	FUNCTION_BLOCK FB 1042
	TITLE =A_2914_MXZ01MA BELT CONVEYOR 4600 GERM 3
	//COPYRIGHT:     (C) 2009  BUHLER AG, CH-9240 UZWIL, SWITZERLAND
	//
	//PRODUCT:       WinCoS_BIW01_09
	//
	//TITLE:         BELT CONVEYOR 4600 GERM 3
	//
	//--------------------------------------------------------------------------------
	//
	//IDENT:         AUTHOR:             DEPT:                             DATE:
	//
	//P01_FB1042.1.0 K.Renz              CSB41                             13.Jan.2010
	//               1st Release
	//
	//--------------------------------------------------------------------------------
	//
	//PURPOSE:
	//
	//MANUAL :
	//
	//RESTRICTIONS:
	//
	//--------------------------------------------------------------------------------
	AUTHOR  : KR
	FAMILY  : USW
	VERSION : 0.0


	VAR
	         Ma :  UDT 20500  ;  // Machine
	         A_2914_SHE41 : FB14;  // Mon1: DigInpCont
	         A_2914_BSA13 : FB14;  // Mon2: DigInpCont
	         A_2914_BZS14_15 : FB14;  // Mon3: DigInpCont
	         A_2914_BZS16_17 : FB14;  // Mon4: DigInpCont
	         A_2914_SHE43 : FB14;  // Mon5: DigInpCont
	         A_2914_SHE44 : FB14;   // Mon6: DigInpCont
	         A_2914_MXZ01 : FB12; // Motor: Motor
	END_VAR

	BEGIN
	NETWORK
	TITLE =Call SSW
	   UC  FB50
	END_FUNCTION_BLOCK
